// TIA Portal V17 program export: 0 tag tables, 0 data types, 0 data blocks, 5 code blocks (in call order from the OBs), 0 instance data blocks

ORGANIZATION_BLOCK "OB1_CYCLE"   // OB1, LAD, ProgramCycle
TITLE = "Main Program Sweep (Cycle)"
{ S7_Optimized_Access := 'FALSE' }
AUTHOR : ETXETAR
VERSION : 1.0
// stored: AutoNumber false, IsIECCheckEnabled false, SetENOAutomatically false
   VAR_TEMP
      OB1_SCAN : Byte;   // 1 (Cold restart scan 1 of OB 1), 3 (Scan 2-n of OB 1)
      OB1_PRIORITY : Int;   // Priority of OB Execution
      OB1_MIN_CYCLE : DInt;   // Minimum cycle time of OB1 (milliseconds)
      OB1_MAX_CYCLE : DInt;   // Maximum cycle time of OB1 (milliseconds)
      PART_TYPE : Int;
      zero : Byte;
      status_sfc21 : Int;
      Error : Bool;
      status : Word;
   END_VAR
   VAR_TEMP   // added for the SCL form of the ladder/FBD networks
      _w1 : Bool;
   END_VAR
BEGIN

REGION Network 1: CALL FC2
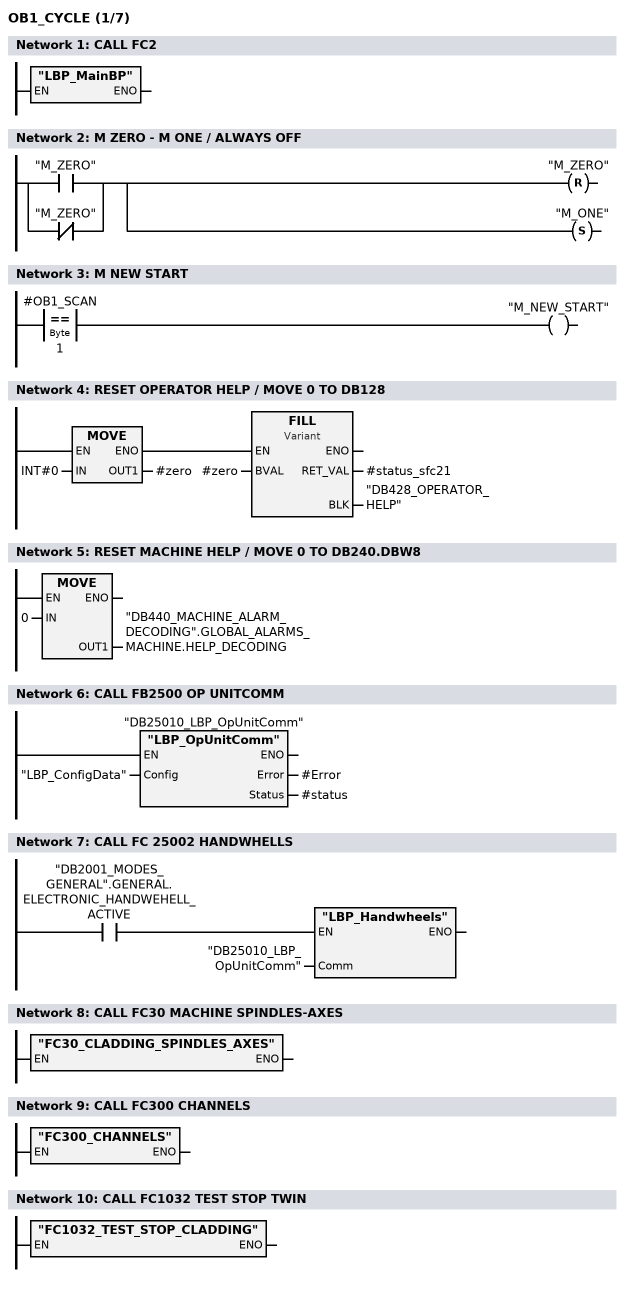
   RUNG wire#powerrail
      "LBP_MainBP"()
   END_RUNG
   // the same network as SCL:
   "LBP_MainBP"();
END_REGION

REGION Network 2: M ZERO - M ONE / ALWAYS OFF
   RUNG wire#powerrail
      Contact( "M_ZERO" )
      wire#w1
      R_Coil( "M_ZERO" )
   END_RUNG
   RUNG wire#powerrail
      I_Contact( "M_ZERO" )
   END_RUNG wire#w1
   RUNG wire#w1
      S_Coil( "M_ONE" )
   END_RUNG
   // the same network as SCL:
   #_w1 := "M_ZERO" OR NOT "M_ZERO";
   IF #_w1 THEN
       "M_ZERO" := FALSE;
       "M_ONE" := TRUE;
   END_IF;
END_REGION

REGION Network 3: M NEW START
   RUNG wire#powerrail
      { S7_Templates := "SrcType := Byte" } EQ_Contact(in1 := #OB1_SCAN, in2 := 1)
      Coil( "M_NEW_START" )
   END_RUNG
   // the same network as SCL:
   "M_NEW_START" := #OB1_SCAN = 1;
END_REGION

REGION Network 4: RESET OPERATOR HELP / MOVE 0 TO DB128
   RUNG wire#powerrail
      { S7_GenerateENO := "TRUE" } Move(in := INT#0, out1 => #zero)
      { S7_Templates := "ptr_type := Variant" } FILL(BVAL := #zero, RET_VAL => #status_sfc21, BLK => "DB428_OPERATOR_HELP")
   END_RUNG
   // the same network as SCL:
   // ENO of a box is taken as its EN; it also drops when the box reports an error
   #zero := INT#0;
   #status_sfc21 := FILL(BVAL := #zero, BLK => "DB428_OPERATOR_HELP");
END_REGION

REGION Network 5: RESET MACHINE HELP / MOVE 0 TO DB240.DBW8
   RUNG wire#powerrail
      { S7_GenerateENO := "TRUE" } Move(in := 0, out1 => "DB440_MACHINE_ALARM_DECODING".GLOBAL_ALARMS_MACHINE.HELP_DECODING)
   END_RUNG
   // the same network as SCL:
   "DB440_MACHINE_ALARM_DECODING".GLOBAL_ALARMS_MACHINE.HELP_DECODING := 0;
END_REGION

REGION Network 6: CALL FB2500 OP UNITCOMM
   RUNG wire#powerrail
      "DB25010_LBP_OpUnitComm"(Config := "LBP_ConfigData", Error => #Error, Status => #status)
   END_RUNG
   // the same network as SCL:
   "DB25010_LBP_OpUnitComm"(Config := "LBP_ConfigData", Error => #Error, Status => #status);   // "LBP_OpUnitComm"
END_REGION

REGION Network 7: CALL FC 25002 HANDWHELLS
   RUNG wire#powerrail
      Contact( "DB2001_MODES_GENERAL".GENERAL.ELECTRONIC_HANDWEHELL_ACTIVE )
      "LBP_Handwheels"(Comm := "DB25010_LBP_OpUnitComm")
   END_RUNG
   // the same network as SCL:
   IF "DB2001_MODES_GENERAL".GENERAL.ELECTRONIC_HANDWEHELL_ACTIVE THEN
       "LBP_Handwheels"(Comm := "DB25010_LBP_OpUnitComm");
   END_IF;
END_REGION

REGION Network 8: CALL FC30 MACHINE SPINDLES-AXES
   RUNG wire#powerrail
      "FC30_CLADDING_SPINDLES_AXES"()
   END_RUNG
   // the same network as SCL:
   "FC30_CLADDING_SPINDLES_AXES"();
END_REGION

REGION Network 9: CALL FC300 CHANNELS
   RUNG wire#powerrail
      "FC300_CHANNELS"()
   END_RUNG
   // the same network as SCL:
   "FC300_CHANNELS"();
END_REGION

REGION Network 10: CALL FC1032 TEST STOP TWIN
   RUNG wire#powerrail
      "FC1032_TEST_STOP_CLADDING"()
   END_RUNG
   // the same network as SCL:
   "FC1032_TEST_STOP_CLADDING"();
END_REGION

REGION Network 11: CALL FC1090 IDEVICE SI
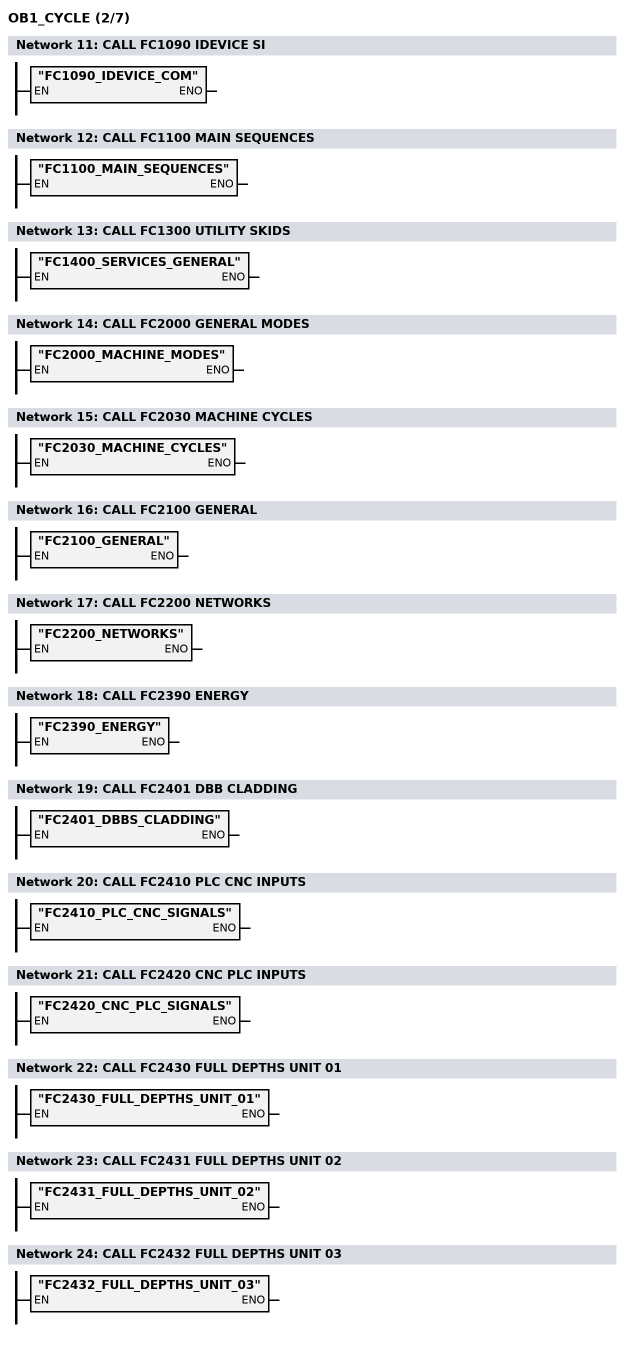
   RUNG wire#powerrail
      "FC1090_IDEVICE_COM"()
   END_RUNG
   // the same network as SCL:
   "FC1090_IDEVICE_COM"();
END_REGION

REGION Network 12: CALL FC1100 MAIN SEQUENCES
   RUNG wire#powerrail
      "FC1100_MAIN_SEQUENCES"()
   END_RUNG
   // the same network as SCL:
   "FC1100_MAIN_SEQUENCES"();
END_REGION

REGION Network 13: CALL FC1300 UTILITY SKIDS
   RUNG wire#powerrail
      "FC1400_SERVICES_GENERAL"()
   END_RUNG
   // the same network as SCL:
   "FC1400_SERVICES_GENERAL"();
END_REGION

REGION Network 14: CALL FC2000 GENERAL MODES
   RUNG wire#powerrail
      "FC2000_MACHINE_MODES"()
   END_RUNG
   // the same network as SCL:
   "FC2000_MACHINE_MODES"();
END_REGION

REGION Network 15: CALL FC2030 MACHINE CYCLES
   RUNG wire#powerrail
      "FC2030_MACHINE_CYCLES"()
   END_RUNG
   // the same network as SCL:
   "FC2030_MACHINE_CYCLES"();
END_REGION

REGION Network 16: CALL FC2100 GENERAL
   RUNG wire#powerrail
      "FC2100_GENERAL"()
   END_RUNG
   // the same network as SCL:
   "FC2100_GENERAL"();
END_REGION

REGION Network 17: CALL FC2200 NETWORKS
   RUNG wire#powerrail
      "FC2200_NETWORKS"()
   END_RUNG
   // the same network as SCL:
   "FC2200_NETWORKS"();
END_REGION

REGION Network 18: CALL FC2390 ENERGY
   RUNG wire#powerrail
      "FC2390_ENERGY"()
   END_RUNG
   // the same network as SCL:
   "FC2390_ENERGY"();
END_REGION

REGION Network 19: CALL FC2401 DBB CLADDING
   RUNG wire#powerrail
      "FC2401_DBBS_CLADDING"()
   END_RUNG
   // the same network as SCL:
   "FC2401_DBBS_CLADDING"();
END_REGION

REGION Network 20: CALL FC2410 PLC CNC INPUTS
   RUNG wire#powerrail
      "FC2410_PLC_CNC_SIGNALS"()
   END_RUNG
   // the same network as SCL:
   "FC2410_PLC_CNC_SIGNALS"();
END_REGION

REGION Network 21: CALL FC2420 CNC PLC INPUTS
   RUNG wire#powerrail
      "FC2420_CNC_PLC_SIGNALS"()
   END_RUNG
   // the same network as SCL:
   "FC2420_CNC_PLC_SIGNALS"();
END_REGION

REGION Network 22: CALL FC2430 FULL DEPTHS UNIT 01
   RUNG wire#powerrail
      "FC2430_FULL_DEPTHS_UNIT_01"()
   END_RUNG
   // the same network as SCL:
   "FC2430_FULL_DEPTHS_UNIT_01"();
END_REGION

REGION Network 23: CALL FC2431 FULL DEPTHS UNIT 02
   RUNG wire#powerrail
      "FC2431_FULL_DEPTHS_UNIT_02"()
   END_RUNG
   // the same network as SCL:
   "FC2431_FULL_DEPTHS_UNIT_02"();
END_REGION

REGION Network 24: CALL FC2432 FULL DEPTHS UNIT 03
   RUNG wire#powerrail
      "FC2432_FULL_DEPTHS_UNIT_03"()
   END_RUNG
   // the same network as SCL:
   "FC2432_FULL_DEPTHS_UNIT_03"();
END_REGION

REGION Network 25: CALL FC2440 GLOBAL DATA CLADDING
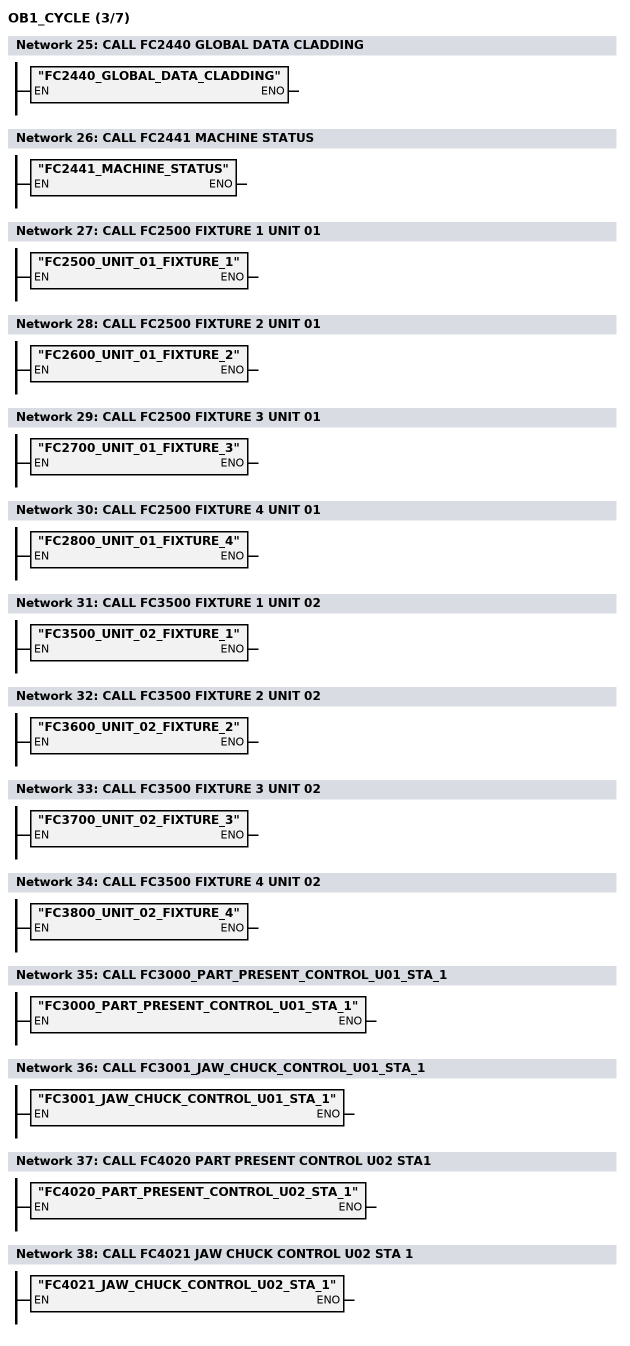
   RUNG wire#powerrail
      "FC2440_GLOBAL_DATA_CLADDING"()
   END_RUNG
   // the same network as SCL:
   "FC2440_GLOBAL_DATA_CLADDING"();
END_REGION

REGION Network 26: CALL FC2441 MACHINE STATUS
   RUNG wire#powerrail
      "FC2441_MACHINE_STATUS"()
   END_RUNG
   // the same network as SCL:
   "FC2441_MACHINE_STATUS"();
END_REGION

REGION Network 27: CALL FC2500 FIXTURE 1 UNIT 01
   RUNG wire#powerrail
      "FC2500_UNIT_01_FIXTURE_1"()
   END_RUNG
   // the same network as SCL:
   "FC2500_UNIT_01_FIXTURE_1"();
END_REGION

REGION Network 28: CALL FC2500 FIXTURE 2 UNIT 01
   RUNG wire#powerrail
      "FC2600_UNIT_01_FIXTURE_2"()
   END_RUNG
   // the same network as SCL:
   "FC2600_UNIT_01_FIXTURE_2"();
END_REGION

REGION Network 29: CALL FC2500 FIXTURE 3 UNIT 01
   RUNG wire#powerrail
      "FC2700_UNIT_01_FIXTURE_3"()
   END_RUNG
   // the same network as SCL:
   "FC2700_UNIT_01_FIXTURE_3"();
END_REGION

REGION Network 30: CALL FC2500 FIXTURE 4 UNIT 01
   RUNG wire#powerrail
      "FC2800_UNIT_01_FIXTURE_4"()
   END_RUNG
   // the same network as SCL:
   "FC2800_UNIT_01_FIXTURE_4"();
END_REGION

REGION Network 31: CALL FC3500 FIXTURE 1 UNIT 02
   RUNG wire#powerrail
      "FC3500_UNIT_02_FIXTURE_1"()
   END_RUNG
   // the same network as SCL:
   "FC3500_UNIT_02_FIXTURE_1"();
END_REGION

REGION Network 32: CALL FC3500 FIXTURE 2 UNIT 02
   RUNG wire#powerrail
      "FC3600_UNIT_02_FIXTURE_2"()
   END_RUNG
   // the same network as SCL:
   "FC3600_UNIT_02_FIXTURE_2"();
END_REGION

REGION Network 33: CALL FC3500 FIXTURE 3 UNIT 02
   RUNG wire#powerrail
      "FC3700_UNIT_02_FIXTURE_3"()
   END_RUNG
   // the same network as SCL:
   "FC3700_UNIT_02_FIXTURE_3"();
END_REGION

REGION Network 34: CALL FC3500 FIXTURE 4 UNIT 02
   RUNG wire#powerrail
      "FC3800_UNIT_02_FIXTURE_4"()
   END_RUNG
   // the same network as SCL:
   "FC3800_UNIT_02_FIXTURE_4"();
END_REGION

REGION Network 35: CALL FC3000_PART_PRESENT_CONTROL_U01_STA_1
   RUNG wire#powerrail
      "FC3000_PART_PRESENT_CONTROL_U01_STA_1"()
   END_RUNG
   // the same network as SCL:
   "FC3000_PART_PRESENT_CONTROL_U01_STA_1"();
END_REGION

REGION Network 36: CALL FC3001_JAW_CHUCK_CONTROL_U01_STA_1
   RUNG wire#powerrail
      "FC3001_JAW_CHUCK_CONTROL_U01_STA_1"()
   END_RUNG
   // the same network as SCL:
   "FC3001_JAW_CHUCK_CONTROL_U01_STA_1"();
END_REGION

REGION Network 37: CALL FC4020 PART PRESENT CONTROL U02 STA1
   RUNG wire#powerrail
      "FC4020_PART_PRESENT_CONTROL_U02_STA_1"()
   END_RUNG
   // the same network as SCL:
   "FC4020_PART_PRESENT_CONTROL_U02_STA_1"();
END_REGION

REGION Network 38: CALL FC4021 JAW CHUCK CONTROL U02 STA 1
   RUNG wire#powerrail
      "FC4021_JAW_CHUCK_CONTROL_U02_STA_1"()
   END_RUNG
   // the same network as SCL:
   "FC4021_JAW_CHUCK_CONTROL_U02_STA_1"();
END_REGION

REGION Network 39: CALL FC4000 FIXTURE TABLE POSITIONS
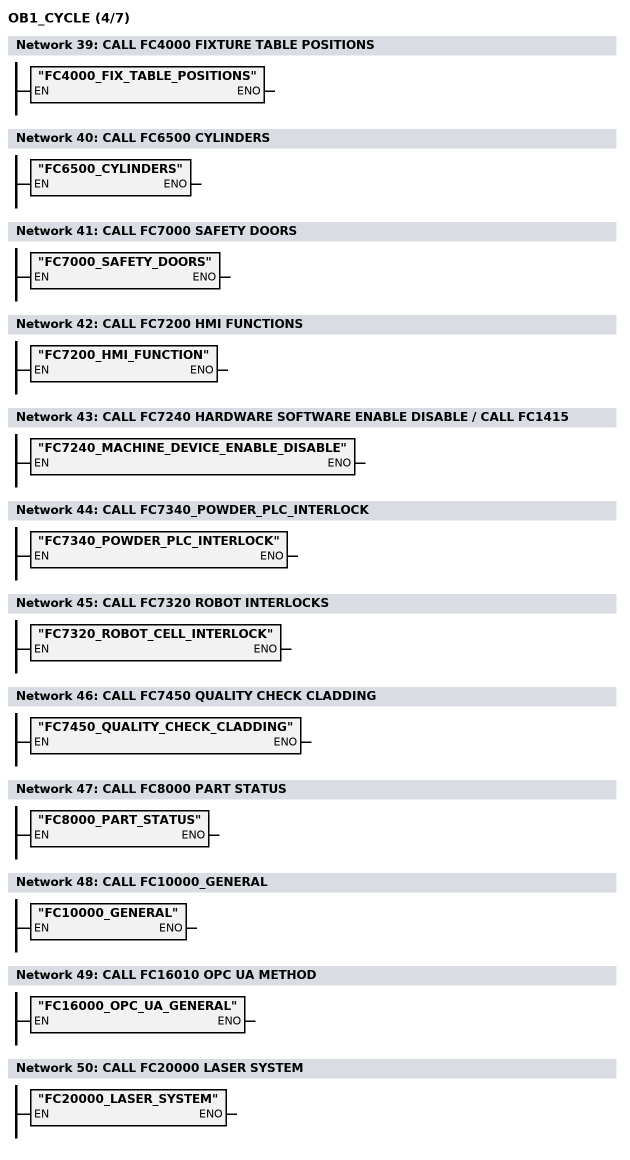
   RUNG wire#powerrail
      "FC4000_FIX_TABLE_POSITIONS"()
   END_RUNG
   // the same network as SCL:
   "FC4000_FIX_TABLE_POSITIONS"();
END_REGION

REGION Network 40: CALL FC6500 CYLINDERS
   RUNG wire#powerrail
      "FC6500_CYLINDERS"()
   END_RUNG
   // the same network as SCL:
   "FC6500_CYLINDERS"();
END_REGION

REGION Network 41: CALL FC7000 SAFETY DOORS
   RUNG wire#powerrail
      "FC7000_SAFETY_DOORS"()
   END_RUNG
   // the same network as SCL:
   "FC7000_SAFETY_DOORS"();
END_REGION

REGION Network 42: CALL FC7200 HMI FUNCTIONS
   RUNG wire#powerrail
      "FC7200_HMI_FUNCTION"()
   END_RUNG
   // the same network as SCL:
   "FC7200_HMI_FUNCTION"();
END_REGION

REGION Network 43: CALL FC7240 HARDWARE SOFTWARE ENABLE DISABLE / CALL FC1415
   RUNG wire#powerrail
      "FC7240_MACHINE_DEVICE_ENABLE_DISABLE"()
   END_RUNG
   // the same network as SCL:
   "FC7240_MACHINE_DEVICE_ENABLE_DISABLE"();
END_REGION

REGION Network 44: CALL FC7340_POWDER_PLC_INTERLOCK
   RUNG wire#powerrail
      "FC7340_POWDER_PLC_INTERLOCK"()
   END_RUNG
   // the same network as SCL:
   "FC7340_POWDER_PLC_INTERLOCK"();
END_REGION

REGION Network 45: CALL FC7320 ROBOT INTERLOCKS
   RUNG wire#powerrail
      "FC7320_ROBOT_CELL_INTERLOCK"()
   END_RUNG
   // the same network as SCL:
   "FC7320_ROBOT_CELL_INTERLOCK"();
END_REGION

REGION Network 46: CALL FC7450 QUALITY CHECK CLADDING
   RUNG wire#powerrail
      "FC7450_QUALITY_CHECK_CLADDING"()
   END_RUNG
   // the same network as SCL:
   "FC7450_QUALITY_CHECK_CLADDING"();
END_REGION

REGION Network 47: CALL FC8000 PART STATUS
   RUNG wire#powerrail
      "FC8000_PART_STATUS"()
   END_RUNG
   // the same network as SCL:
   "FC8000_PART_STATUS"();
END_REGION

REGION Network 48: CALL FC10000_GENERAL
   RUNG wire#powerrail
      "FC10000_GENERAL"()
   END_RUNG
   // the same network as SCL:
   "FC10000_GENERAL"();
END_REGION

REGION Network 49: CALL FC16010 OPC UA METHOD
   RUNG wire#powerrail
      "FC16000_OPC_UA_GENERAL"()
   END_RUNG
   // the same network as SCL:
   "FC16000_OPC_UA_GENERAL"();
END_REGION

REGION Network 50: CALL FC20000 LASER SYSTEM
   RUNG wire#powerrail
      "FC20000_LASER_SYSTEM"()
   END_RUNG
   // the same network as SCL:
   "FC20000_LASER_SYSTEM"();
END_REGION

REGION Network 51: SCREEN DARKENING
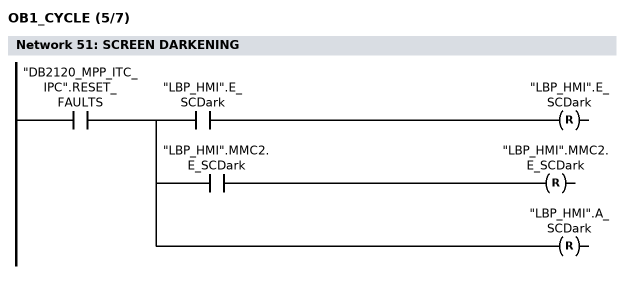
   RUNG wire#powerrail
      Contact( "DB2120_MPP_ITC_IPC".RESET_FAULTS )
      wire#w1
      Contact( "LBP_HMI".E_SCDark )
      R_Coil( "LBP_HMI".E_SCDark )
   END_RUNG
   RUNG wire#w1
      Contact( "LBP_HMI".MMC2.E_SCDark )
      R_Coil( "LBP_HMI".MMC2.E_SCDark )
   END_RUNG
   RUNG wire#w1
      R_Coil( "LBP_HMI".A_SCDark )
   END_RUNG
   // the same network as SCL:
   IF "DB2120_MPP_ITC_IPC".RESET_FAULTS AND "LBP_HMI".E_SCDark THEN "LBP_HMI".E_SCDark := FALSE; END_IF;
   IF "DB2120_MPP_ITC_IPC".RESET_FAULTS AND "LBP_HMI".MMC2.E_SCDark THEN
       "LBP_HMI".MMC2.E_SCDark := FALSE;
   END_IF;
   IF "DB2120_MPP_ITC_IPC".RESET_FAULTS THEN "LBP_HMI".A_SCDark := FALSE; END_IF;
END_REGION

REGION Network 52: OPERATOR HELP
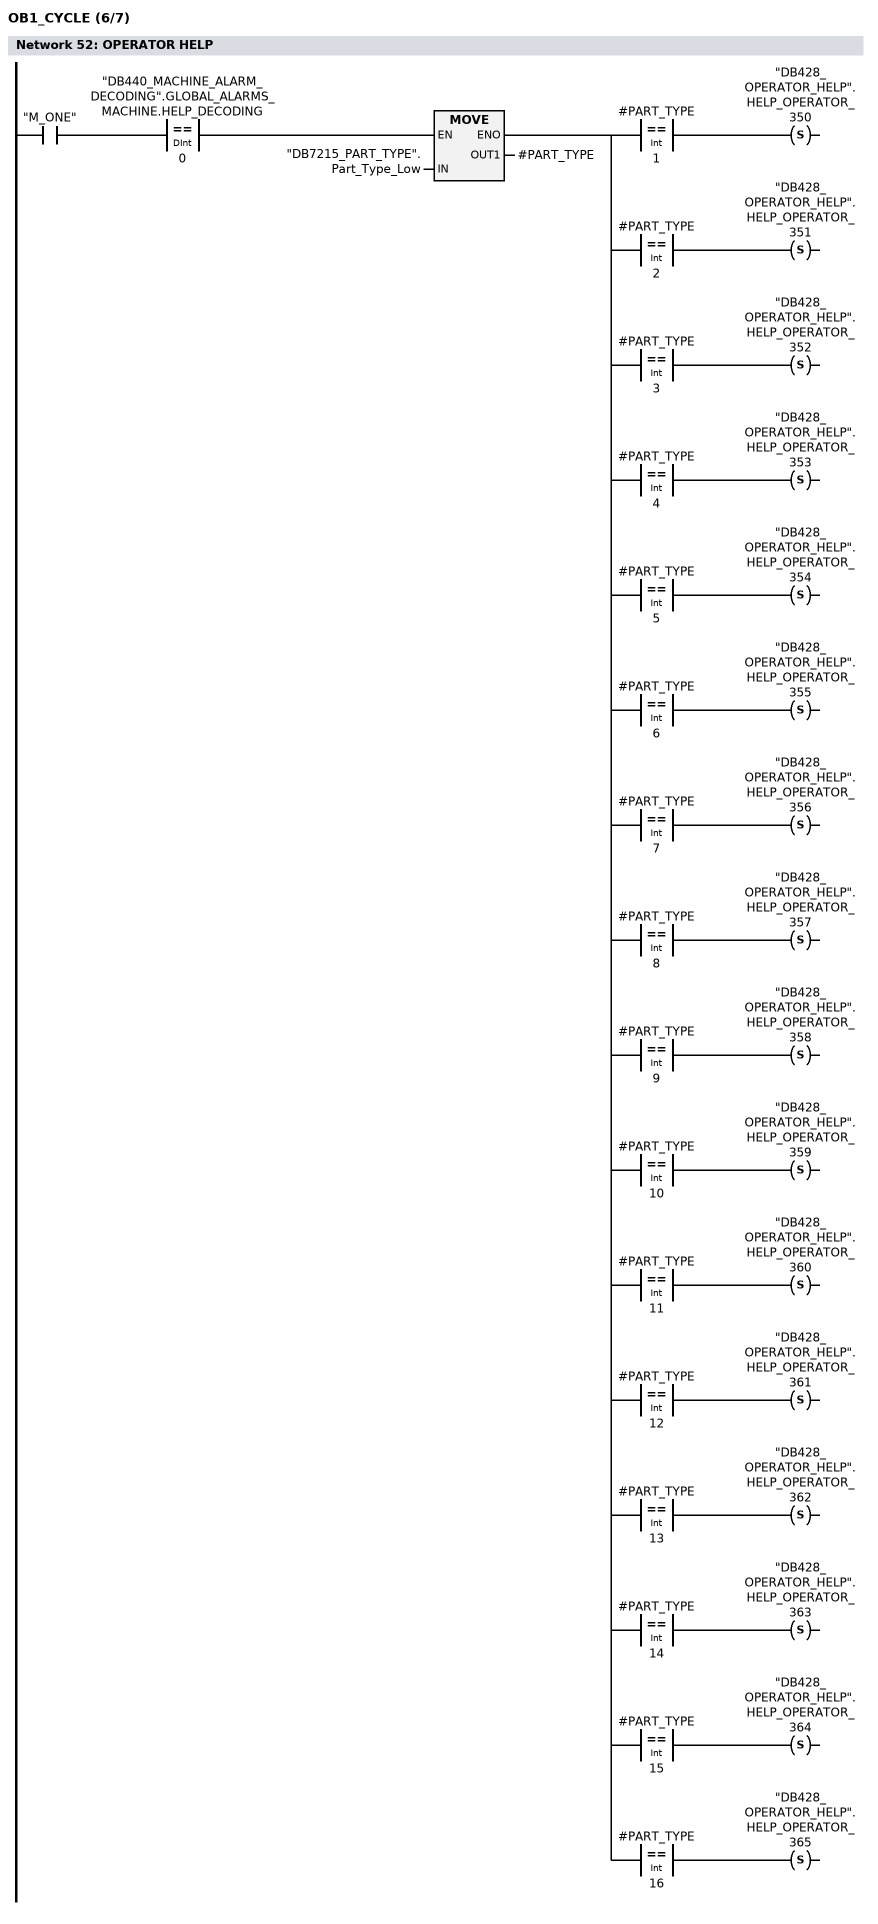
   RUNG wire#powerrail
      Contact( "M_ONE" )
      { S7_Templates := "SrcType := DInt" } EQ_Contact(in1 := "DB440_MACHINE_ALARM_DECODING".GLOBAL_ALARMS_MACHINE.HELP_DECODING, in2 := 0)
      { S7_GenerateENO := "TRUE" } Move(in := "DB7215_PART_TYPE".Part_Type_Low, out1 => #PART_TYPE)
      wire#w1
      { S7_Templates := "SrcType := Int" } EQ_Contact(in1 := #PART_TYPE, in2 := 1)
      S_Coil( "DB428_OPERATOR_HELP".HELP_OPERATOR_350 )
   END_RUNG
   RUNG wire#w1
      { S7_Templates := "SrcType := Int" } EQ_Contact(in1 := #PART_TYPE, in2 := 2)
      S_Coil( "DB428_OPERATOR_HELP".HELP_OPERATOR_351 )
   END_RUNG
   RUNG wire#w1
      { S7_Templates := "SrcType := Int" } EQ_Contact(in1 := #PART_TYPE, in2 := 3)
      S_Coil( "DB428_OPERATOR_HELP".HELP_OPERATOR_352 )
   END_RUNG
   RUNG wire#w1
      { S7_Templates := "SrcType := Int" } EQ_Contact(in1 := #PART_TYPE, in2 := 4)
      S_Coil( "DB428_OPERATOR_HELP".HELP_OPERATOR_353 )
   END_RUNG
   RUNG wire#w1
      { S7_Templates := "SrcType := Int" } EQ_Contact(in1 := #PART_TYPE, in2 := 5)
      S_Coil( "DB428_OPERATOR_HELP".HELP_OPERATOR_354 )
   END_RUNG
   RUNG wire#w1
      { S7_Templates := "SrcType := Int" } EQ_Contact(in1 := #PART_TYPE, in2 := 6)
      S_Coil( "DB428_OPERATOR_HELP".HELP_OPERATOR_355 )
   END_RUNG
   RUNG wire#w1
      { S7_Templates := "SrcType := Int" } EQ_Contact(in1 := #PART_TYPE, in2 := 7)
      S_Coil( "DB428_OPERATOR_HELP".HELP_OPERATOR_356 )
   END_RUNG
   RUNG wire#w1
      { S7_Templates := "SrcType := Int" } EQ_Contact(in1 := #PART_TYPE, in2 := 8)
      S_Coil( "DB428_OPERATOR_HELP".HELP_OPERATOR_357 )
   END_RUNG
   RUNG wire#w1
      { S7_Templates := "SrcType := Int" } EQ_Contact(in1 := #PART_TYPE, in2 := 9)
      S_Coil( "DB428_OPERATOR_HELP".HELP_OPERATOR_358 )
   END_RUNG
   RUNG wire#w1
      { S7_Templates := "SrcType := Int" } EQ_Contact(in1 := #PART_TYPE, in2 := 10)
      S_Coil( "DB428_OPERATOR_HELP".HELP_OPERATOR_359 )
   END_RUNG
   RUNG wire#w1
      { S7_Templates := "SrcType := Int" } EQ_Contact(in1 := #PART_TYPE, in2 := 11)
      S_Coil( "DB428_OPERATOR_HELP".HELP_OPERATOR_360 )
   END_RUNG
   RUNG wire#w1
      { S7_Templates := "SrcType := Int" } EQ_Contact(in1 := #PART_TYPE, in2 := 12)
      S_Coil( "DB428_OPERATOR_HELP".HELP_OPERATOR_361 )
   END_RUNG
   RUNG wire#w1
      { S7_Templates := "SrcType := Int" } EQ_Contact(in1 := #PART_TYPE, in2 := 13)
      S_Coil( "DB428_OPERATOR_HELP".HELP_OPERATOR_362 )
   END_RUNG
   RUNG wire#w1
      { S7_Templates := "SrcType := Int" } EQ_Contact(in1 := #PART_TYPE, in2 := 14)
      S_Coil( "DB428_OPERATOR_HELP".HELP_OPERATOR_363 )
   END_RUNG
   RUNG wire#w1
      { S7_Templates := "SrcType := Int" } EQ_Contact(in1 := #PART_TYPE, in2 := 15)
      S_Coil( "DB428_OPERATOR_HELP".HELP_OPERATOR_364 )
   END_RUNG
   RUNG wire#w1
      { S7_Templates := "SrcType := Int" } EQ_Contact(in1 := #PART_TYPE, in2 := 16)
      S_Coil( "DB428_OPERATOR_HELP".HELP_OPERATOR_365 )
   END_RUNG
   // the same network as SCL:
   // ENO of a box is taken as its EN; it also drops when the box reports an error
   #_w1 := "M_ONE" AND ("DB440_MACHINE_ALARM_DECODING".GLOBAL_ALARMS_MACHINE.HELP_DECODING = 0);
   IF #_w1 THEN #PART_TYPE := "DB7215_PART_TYPE".Part_Type_Low; END_IF;
   IF #_w1 AND (#PART_TYPE = 1) THEN "DB428_OPERATOR_HELP".HELP_OPERATOR_350 := TRUE; END_IF;
   IF #_w1 AND (#PART_TYPE = 2) THEN "DB428_OPERATOR_HELP".HELP_OPERATOR_351 := TRUE; END_IF;
   IF #_w1 AND (#PART_TYPE = 3) THEN "DB428_OPERATOR_HELP".HELP_OPERATOR_352 := TRUE; END_IF;
   IF #_w1 AND (#PART_TYPE = 4) THEN "DB428_OPERATOR_HELP".HELP_OPERATOR_353 := TRUE; END_IF;
   IF #_w1 AND (#PART_TYPE = 5) THEN "DB428_OPERATOR_HELP".HELP_OPERATOR_354 := TRUE; END_IF;
   IF #_w1 AND (#PART_TYPE = 6) THEN "DB428_OPERATOR_HELP".HELP_OPERATOR_355 := TRUE; END_IF;
   IF #_w1 AND (#PART_TYPE = 7) THEN "DB428_OPERATOR_HELP".HELP_OPERATOR_356 := TRUE; END_IF;
   IF #_w1 AND (#PART_TYPE = 8) THEN "DB428_OPERATOR_HELP".HELP_OPERATOR_357 := TRUE; END_IF;
   IF #_w1 AND (#PART_TYPE = 9) THEN "DB428_OPERATOR_HELP".HELP_OPERATOR_358 := TRUE; END_IF;
   IF #_w1 AND (#PART_TYPE = 10) THEN "DB428_OPERATOR_HELP".HELP_OPERATOR_359 := TRUE; END_IF;
   IF #_w1 AND (#PART_TYPE = 11) THEN "DB428_OPERATOR_HELP".HELP_OPERATOR_360 := TRUE; END_IF;
   IF #_w1 AND (#PART_TYPE = 12) THEN "DB428_OPERATOR_HELP".HELP_OPERATOR_361 := TRUE; END_IF;
   IF #_w1 AND (#PART_TYPE = 13) THEN "DB428_OPERATOR_HELP".HELP_OPERATOR_362 := TRUE; END_IF;
   IF #_w1 AND (#PART_TYPE = 14) THEN "DB428_OPERATOR_HELP".HELP_OPERATOR_363 := TRUE; END_IF;
   IF #_w1 AND (#PART_TYPE = 15) THEN "DB428_OPERATOR_HELP".HELP_OPERATOR_364 := TRUE; END_IF;
   IF #_w1 AND (#PART_TYPE = 16) THEN "DB428_OPERATOR_HELP".HELP_OPERATOR_365 := TRUE; END_IF;
END_REGION

REGION Network 53: CALL FC428 OPERATOR HELP
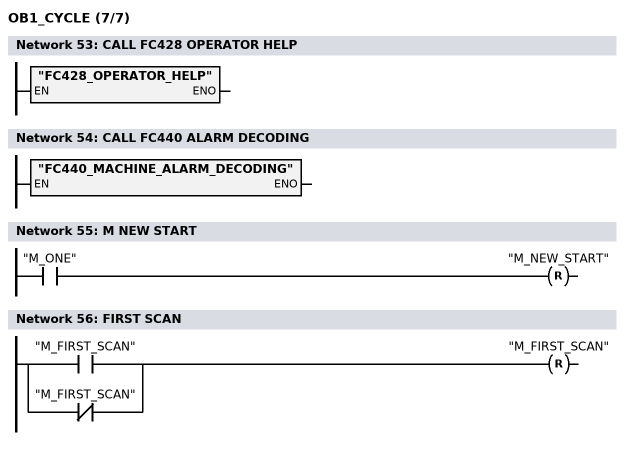
   RUNG wire#powerrail
      "FC428_OPERATOR_HELP"()
   END_RUNG
   // the same network as SCL:
   "FC428_OPERATOR_HELP"();
END_REGION

REGION Network 54: CALL FC440 ALARM DECODING
   RUNG wire#powerrail
      "FC440_MACHINE_ALARM_DECODING"()
   END_RUNG
   // the same network as SCL:
   "FC440_MACHINE_ALARM_DECODING"();
END_REGION

REGION Network 55: M NEW START
   RUNG wire#powerrail
      Contact( "M_ONE" )
      R_Coil( "M_NEW_START" )
   END_RUNG
   // the same network as SCL:
   IF "M_ONE" THEN "M_NEW_START" := FALSE; END_IF;
END_REGION

REGION Network 56: FIRST SCAN
   RUNG wire#powerrail
      Contact( "M_FIRST_SCAN" )
      wire#w1
      R_Coil( "M_FIRST_SCAN" )
   END_RUNG
   RUNG wire#powerrail
      I_Contact( "M_FIRST_SCAN" )
   END_RUNG wire#w1
   // the same network as SCL:
   IF "M_FIRST_SCAN" OR NOT "M_FIRST_SCAN" THEN "M_FIRST_SCAN" := FALSE; END_IF;
END_REGION
END_ORGANIZATION_BLOCK

ORGANIZATION_BLOCK "OB100_RESTART"   // OB100, LAD, Startup
TITLE = "Complete Restart"
{ S7_Optimized_Access := 'FALSE' }
AUTHOR : ETXETAR
VERSION : 1.0
// stored: AutoNumber false, IsIECCheckEnabled false, SetENOAutomatically false
   VAR_TEMP
      OB100_EV_CLASS : Byte;
      OB100_STRTUP : Byte;
      OB100_PRIORITY : Byte;
      OB100_OB_NUMBR : Byte;
      OB100_RESERVED_1 : Byte;
      OB100_RESERVED_2 : Byte;
      OB100_STOP : Word;
      OB100_RESERVED_3 : Word;
      OB100_RESERVED_4 : Word;
      OB100_DATE_TIME : Date_And_Time;
      __PlcmigTempFillBits_20B0 : Array[0..7] of Bool;
   END_VAR
BEGIN

REGION Network 1: M_ONE / ESTABLISH "LOGIC 1" BIT
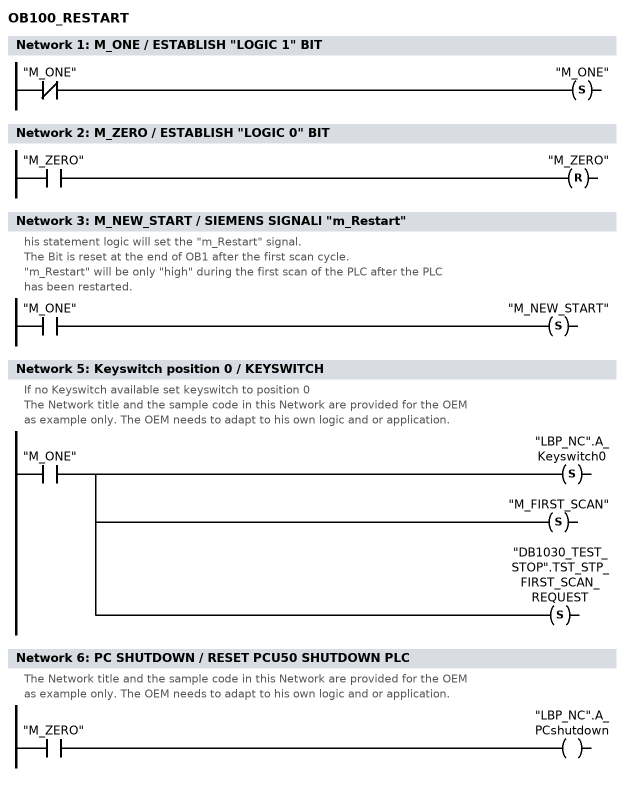
   RUNG wire#powerrail
      I_Contact( "M_ONE" )
      S_Coil( "M_ONE" )
   END_RUNG
   // the same network as SCL:
   IF NOT "M_ONE" THEN "M_ONE" := TRUE; END_IF;
END_REGION

REGION Network 2: M_ZERO / ESTABLISH "LOGIC 0" BIT
   RUNG wire#powerrail
      Contact( "M_ZERO" )
      R_Coil( "M_ZERO" )
   END_RUNG
   // the same network as SCL:
   IF "M_ZERO" THEN "M_ZERO" := FALSE; END_IF;
END_REGION

REGION Network 3: M_NEW_START / SIEMENS SIGNALl "m_Restart"
   // his statement logic will set the "m_Restart" signal.
   // The Bit is reset at the end of OB1 after the first scan cycle.
   // 
   // "m_Restart" will be only "high" during the first scan of the PLC after the PLC 
   // has been restarted.
   RUNG wire#powerrail
      Contact( "M_ONE" )
      S_Coil( "M_NEW_START" )
   END_RUNG
   // the same network as SCL:
   IF "M_ONE" THEN "M_NEW_START" := TRUE; END_IF;
END_REGION

NETWORK
TITLE = CALL FC1
      CALL  "LBP_ConfigBP"
      ( MCPNum             := 2,
        MCP1In             := "MPP_INS",
        MCP1Out            := "MPP_OUT",
        MCP1BusAdr         := 192,
        MCP1Timeout        := S5T#700MS,
        MCP2In             := "HT10_INS",
        MCP2Out            := "HT10_OUTS",
        MCP2BusAdr         := 14,
        MCP2Timeout        := S5T#700MS,
        MCP1Stop           := FALSE,
        MCP2Stop           := FALSE,
        MCP1NotSend        := FALSE,
        MCP2NotSend        := FALSE,
        MCPBusType         := B#16#55,
        HTIf               := 0,
        HTIn               := NULL,
        HTOut              := NULL,
        HTAdr              := 2,
        HTStop             := FALSE,
        HTNotSend          := FALSE,
        NCCyclTimeout      := S5T#200MS,
        NCRunupTimeout     := S5T#50S,
        ListMDecGrp        := 0,
        MMCToIF            := TRUE,
        HWheelMMC          := FALSE,
        MCP_IF_TCS         := FALSE,
        ExtendChanAxMsg    := FALSE,
        HMIAxisSel         := FALSE,
        MsgUser            := 10,
        IRAuxfuT           := FALSE,
        IRAuxfuH           := FALSE,
        IRAuxfuE           := FALSE,
        UserVersion        := "LBP_ConfigData".UserVersionInfo,
        OpKeyNum           := 0,
        Op1KeyIn           := NULL,
        Op1KeyOut          := NULL,
        Op1KeyBusAdr       := 0,
        Op2KeyIn           := NULL,
        Op2KeyOut          := NULL,
        Op2KeyBusAdr       := 0,
        Op1KeyStop         := FALSE,
        Op2KeyStop         := FALSE,
        Op1KeyNotSend      := FALSE,
        Op2KeyNotSend      := FALSE,
        OpUnitCommId       := 1,
        OpUnitInterfaceId  := 262,
        MCP1ConnectionId   := 1001,
        MCP2ConnectionId   := 1002,
        HTConnectionId     := 1003,
        Op1KeyConnectionId := 1004,
        Op2KeyConnectionId := 1005,
        IdentConnectionId  := 1006,
        MCP1LocalUdpPort   := 16001,
        MCP2LocalUdpPort   := 16002,
        HTLocalUdpPort     := 16003,
        Op1KeyLocalUdpPort := 16004,
        Op2KeyLocalUdpPort := 16005,
        IdentLocalUdpPort  := 16006,
        MaxModeGroup       := "LBP_ConfigData".MaxModeGroup,
        MaxChan            := "LBP_ConfigData".MaxChan,
        MaxAxis            := "LBP_ConfigData".MaxAxis,
        ActiveChan         := "LBP_ConfigData".ActiveChan,
        ActiveAxis         := "LBP_ConfigData".ActiveAxis,
        MaxNumUserDataInt  := "LBP_ConfigData".MaxNumUserDataInt,
        MaxNumUserDataHex  := "LBP_ConfigData".MaxNumUserDataHex,
        MaxNumUserDataReal := "LBP_ConfigData".MaxNumUserDataReal,
        UserDataIntArray   := NULL,
        UserDataHexArray   := NULL,
        UserDataRealArray  := NULL,
        TMMagazines        := NULL
      );







REGION Network 5: Keyswitch position 0 / KEYSWITCH
   // If no Keyswitch available set keyswitch to position 0
   // 
   // The Network title and the sample code in this Network are provided for the OEM 
   // as example only. The OEM needs to adapt to his own logic and or application.
   RUNG wire#powerrail
      Contact( "M_ONE" )
      wire#w1
      S_Coil( "LBP_NC".A_Keyswitch0 )
   END_RUNG
   RUNG wire#w1
      S_Coil( "M_FIRST_SCAN" )
   END_RUNG
   RUNG wire#w1
      S_Coil( "DB1030_TEST_STOP".TST_STP_FIRST_SCAN_REQUEST )
   END_RUNG
   // the same network as SCL:
   IF "M_ONE" THEN
       "LBP_NC".A_Keyswitch0 := TRUE;
       "M_FIRST_SCAN" := TRUE;
       "DB1030_TEST_STOP".TST_STP_FIRST_SCAN_REQUEST := TRUE;
   END_IF;
END_REGION

REGION Network 6: PC SHUTDOWN / RESET PCU50 SHUTDOWN PLC
   // The Network title and the sample code in this Network are provided for the OEM 
   // as example only. The OEM needs to adapt to his own logic and or application.
   RUNG wire#powerrail
      Contact( "M_ZERO" )
      Coil( "LBP_NC".A_PCshutdown )
   END_RUNG
   // the same network as SCL:
   "LBP_NC".A_PCshutdown := "M_ZERO";
END_REGION
END_ORGANIZATION_BLOCK

ORGANIZATION_BLOCK "OB121_SYNCHRONF1"   // OB121, LAD, ProgrammingError
{ S7_Optimized_Access := 'FALSE' }
VERSION : 0.0
// stored: IsIECCheckEnabled false, SetENOAutomatically false
   VAR_TEMP
      TEMP0 : Byte;
      TEMP1 : Byte;
      TEMP2 : Byte;
      TEMP3 : Byte;
      TEMP4 : Byte;
      TEMP5 : Byte;
      TEMP6 : Word;
      TEMP7 : Word;
      TEMP8 : Word;
      TEMP9 : Date_And_Time;
   END_VAR
BEGIN
END_ORGANIZATION_BLOCK

ORGANIZATION_BLOCK "OB122_SYNCHRONF2"   // OB122, LAD, IOAccessError
{ S7_Optimized_Access := 'FALSE' }
VERSION : 0.0
// stored: IsIECCheckEnabled false, SetENOAutomatically false
   VAR_TEMP
      TEMP0 : Byte;
      TEMP1 : Byte;
      TEMP2 : Byte;
      TEMP3 : Byte;
      TEMP4 : Byte;
      TEMP5 : Byte;
      TEMP6 : Word;
      TEMP7 : Word;
      TEMP8 : Word;
      TEMP9 : Date_And_Time;
   END_VAR
BEGIN
END_ORGANIZATION_BLOCK

ORGANIZATION_BLOCK "OB40 Hardware interrupt"   // OB40, LAD, HardwareInterrupt
{ S7_Optimized_Access := 'TRUE' }
VERSION : 0.1
// stored: AutoNumber true, IsIECCheckEnabled false, SetENOAutomatically false
   VAR_INPUT
      LADDR : HW_IO;   // Hardware identifier
      USI : Word;   // User structure identifier
      IChannel : USInt;   // Interrupt channel number
      EventType : Byte;   // EventType
      PointAddr : DWord;
   END_VAR
   VAR_TEMP
      FLAG : Variant;
   END_VAR
BEGIN

REGION Network 2
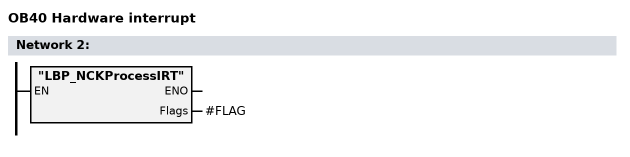
   RUNG wire#powerrail
      "LBP_NCKProcessIRT"(Flags => #FLAG)
   END_RUNG
   // the same network as SCL:
   "LBP_NCKProcessIRT"(Flags => #FLAG);
END_REGION
END_ORGANIZATION_BLOCK
